// Mitsubishi GX Works2 project: 18-06-2020 E10CarparkCounter   PLC: FX3G

PROGRAM MAIN
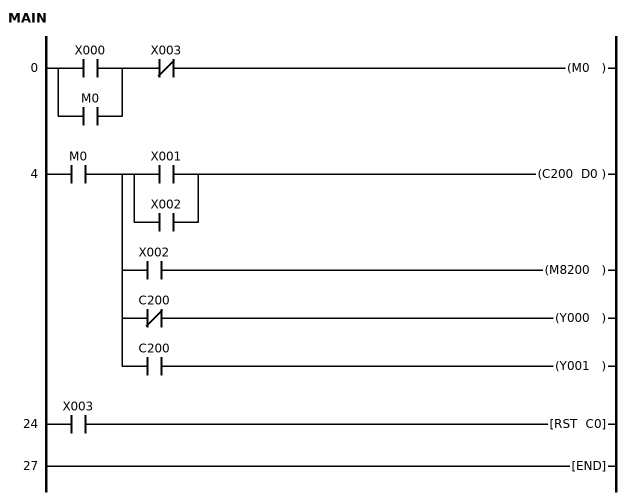
0     LD      X000
      OR      M0
      ANI     X003
      OUT     M0
4     LD      M0
      MPS
      LD      X001
      OR      X002
      ANB
      OUT     C200 D0
      MRD
      AND     X002
      OUT     M8200
      MRD
      ANI     C200
      OUT     Y000
      MPP
      AND     C200
      OUT     Y001
24    LD      X003
      RST     C0
27    END
END_PROGRAM
